// TIA Portal V18 export
FUNCTION_BLOCK "Control_Buttons_Activation"   // FB23, LAD
{ S7_Optimized_Access := 'TRUE' }
VERSION : 0.1
// stored: AutoNumber true, IsIECCheckEnabled false, IsRetainMemResEnabled false, MemoryReserve 100, SetENOAutomatically false, UDAEnableTagReadback false
   VAR_INPUT
      JogInZ1pos : Bool;
      JogInZ1neg : Bool;
      JogInZ2pos : Bool;
      JogInZ2neg : Bool;
   END_VAR
   VAR_OUTPUT
      Control_Buttons_Move_Permission : Bool;
      Control_Buttons_ActivatedOUT : Bool;
   END_VAR
   VAR
      Step01 : Bool;
      Step02 : Bool;
      Step03 : Bool;
      Step04 : Bool;
      Step05 : Bool;
      Step06 : Bool;
      Step07 : Bool;
      Step08 : Bool;
      AnyButtonPressed : Bool;
      AllButtonsPressed : Bool;
      ControlButtonsActivated : Bool;
   END_VAR
BEGIN

REGION Network 1: Any Button Pressed
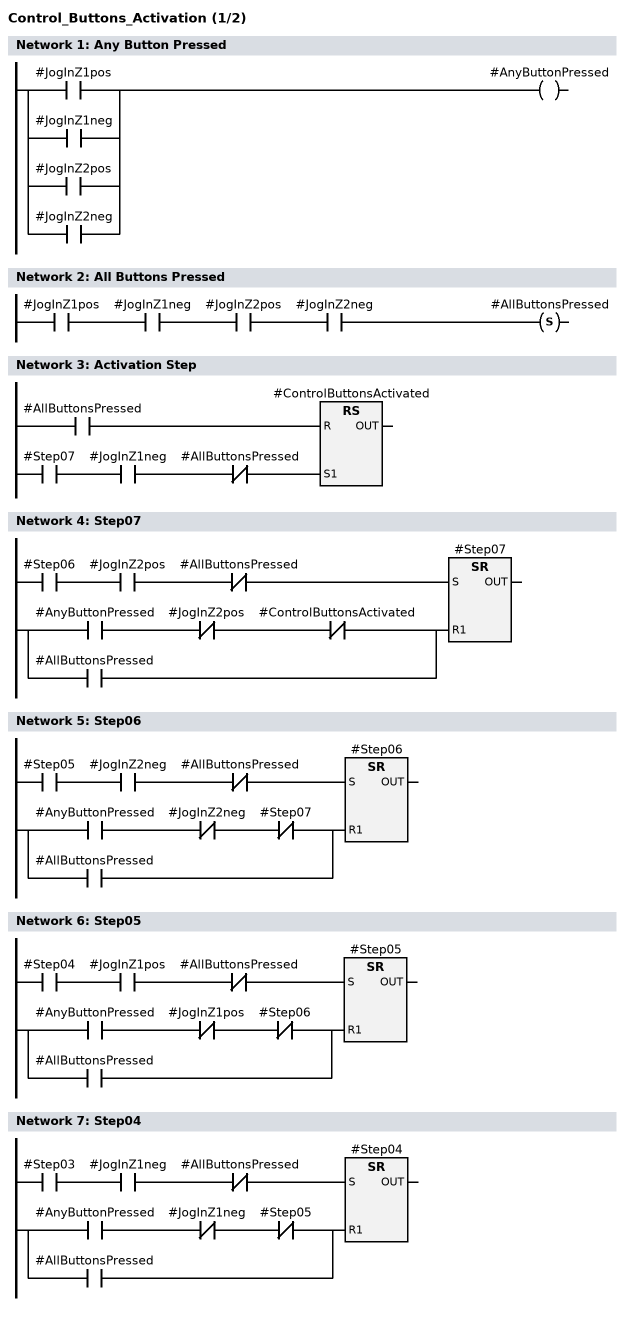
   RUNG wire#powerrail
      Contact( #JogInZ1pos )
      wire#w1
      Coil( #AnyButtonPressed )
   END_RUNG
   RUNG wire#powerrail
      Contact( #JogInZ1neg )
   END_RUNG wire#w1
   RUNG wire#powerrail
      Contact( #JogInZ2pos )
   END_RUNG wire#w1
   RUNG wire#powerrail
      Contact( #JogInZ2neg )
   END_RUNG wire#w1
   // the same network as SCL:
   #AnyButtonPressed := #JogInZ1pos OR #JogInZ1neg OR #JogInZ2pos OR #JogInZ2neg;
END_REGION

REGION Network 2: All Buttons Pressed
   RUNG wire#powerrail
      Contact( #JogInZ1pos )
      Contact( #JogInZ1neg )
      Contact( #JogInZ2pos )
      Contact( #JogInZ2neg )
      S_Coil( #AllButtonsPressed )
   END_RUNG
   // the same network as SCL:
   IF #JogInZ1pos AND #JogInZ1neg AND #JogInZ2pos AND #JogInZ2neg THEN #AllButtonsPressed := TRUE; END_IF;
END_REGION

REGION Network 3: Activation Step
   RUNG wire#powerrail
      Contact( #AllButtonsPressed )
      S_RS(operand := #ControlButtonsActivated, s1 := wire#w1)
   END_RUNG
   RUNG wire#powerrail
      Contact( #Step07 )
      Contact( #JogInZ1neg )
      I_Contact( #AllButtonsPressed )
   END_RUNG wire#w1
   // the same network as SCL:
   IF #AllButtonsPressed THEN
       #ControlButtonsActivated := FALSE;   // RS flip-flop
   END_IF;
   IF #Step07 AND #JogInZ1neg AND NOT #AllButtonsPressed THEN #ControlButtonsActivated := TRUE; END_IF;
END_REGION

REGION Network 4: Step07
   RUNG wire#powerrail
      Contact( #Step06 )
      Contact( #JogInZ2pos )
      I_Contact( #AllButtonsPressed )
      S_SR(operand := #Step07, r1 := wire#w1)
   END_RUNG
   RUNG wire#powerrail
      Contact( #AnyButtonPressed )
      I_Contact( #JogInZ2pos )
      I_Contact( #ControlButtonsActivated )
   END_RUNG wire#w1
   RUNG wire#powerrail
      Contact( #AllButtonsPressed )
   END_RUNG wire#w1
   // the same network as SCL:
   IF #Step06 AND #JogInZ2pos AND NOT #AllButtonsPressed THEN
       #Step07 := TRUE;   // SR flip-flop
   END_IF;
   IF (#AnyButtonPressed AND NOT #JogInZ2pos AND NOT #ControlButtonsActivated) OR #AllButtonsPressed THEN
       #Step07 := FALSE;
   END_IF;
END_REGION

REGION Network 5: Step06
   RUNG wire#powerrail
      Contact( #Step05 )
      Contact( #JogInZ2neg )
      I_Contact( #AllButtonsPressed )
      S_SR(operand := #Step06, r1 := wire#w1)
   END_RUNG
   RUNG wire#powerrail
      Contact( #AnyButtonPressed )
      I_Contact( #JogInZ2neg )
      I_Contact( #Step07 )
   END_RUNG wire#w1
   RUNG wire#powerrail
      Contact( #AllButtonsPressed )
   END_RUNG wire#w1
   // the same network as SCL:
   IF #Step05 AND #JogInZ2neg AND NOT #AllButtonsPressed THEN
       #Step06 := TRUE;   // SR flip-flop
   END_IF;
   IF (#AnyButtonPressed AND NOT #JogInZ2neg AND NOT #Step07) OR #AllButtonsPressed THEN
       #Step06 := FALSE;
   END_IF;
END_REGION

REGION Network 6: Step05
   RUNG wire#powerrail
      Contact( #Step04 )
      Contact( #JogInZ1pos )
      I_Contact( #AllButtonsPressed )
      S_SR(operand := #Step05, r1 := wire#w1)
   END_RUNG
   RUNG wire#powerrail
      Contact( #AnyButtonPressed )
      I_Contact( #JogInZ1pos )
      I_Contact( #Step06 )
   END_RUNG wire#w1
   RUNG wire#powerrail
      Contact( #AllButtonsPressed )
   END_RUNG wire#w1
   // the same network as SCL:
   IF #Step04 AND #JogInZ1pos AND NOT #AllButtonsPressed THEN
       #Step05 := TRUE;   // SR flip-flop
   END_IF;
   IF (#AnyButtonPressed AND NOT #JogInZ1pos AND NOT #Step06) OR #AllButtonsPressed THEN
       #Step05 := FALSE;
   END_IF;
END_REGION

REGION Network 7: Step04
   RUNG wire#powerrail
      Contact( #Step03 )
      Contact( #JogInZ1neg )
      I_Contact( #AllButtonsPressed )
      S_SR(operand := #Step04, r1 := wire#w1)
   END_RUNG
   RUNG wire#powerrail
      Contact( #AnyButtonPressed )
      I_Contact( #JogInZ1neg )
      I_Contact( #Step05 )
   END_RUNG wire#w1
   RUNG wire#powerrail
      Contact( #AllButtonsPressed )
   END_RUNG wire#w1
   // the same network as SCL:
   IF #Step03 AND #JogInZ1neg AND NOT #AllButtonsPressed THEN
       #Step04 := TRUE;   // SR flip-flop
   END_IF;
   IF (#AnyButtonPressed AND NOT #JogInZ1neg AND NOT #Step05) OR #AllButtonsPressed THEN
       #Step04 := FALSE;
   END_IF;
END_REGION

REGION Network 8: Step03
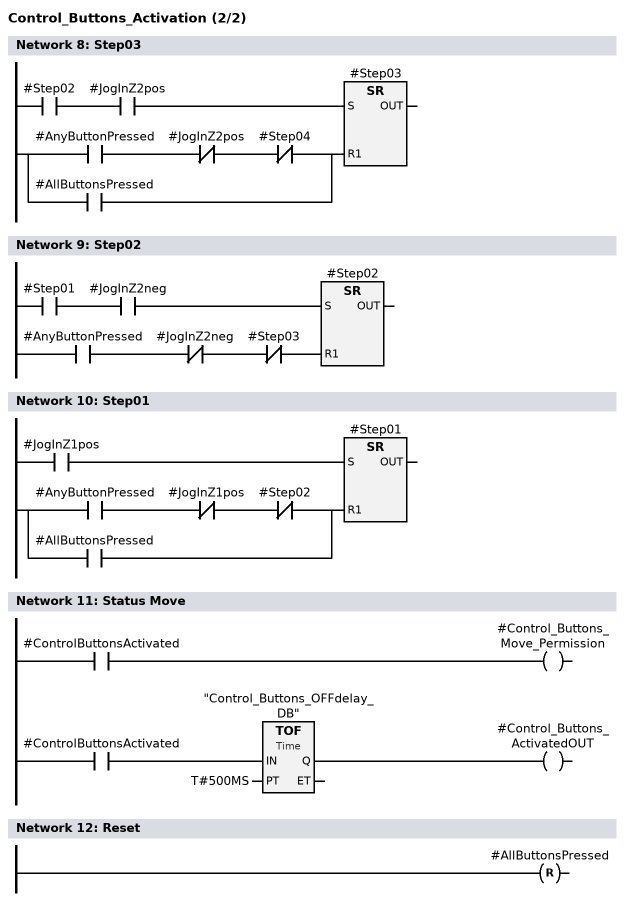
   RUNG wire#powerrail
      Contact( #Step02 )
      Contact( #JogInZ2pos )
      S_SR(operand := #Step03, r1 := wire#w1)
   END_RUNG
   RUNG wire#powerrail
      Contact( #AnyButtonPressed )
      I_Contact( #JogInZ2pos )
      I_Contact( #Step04 )
   END_RUNG wire#w1
   RUNG wire#powerrail
      Contact( #AllButtonsPressed )
   END_RUNG wire#w1
   // the same network as SCL:
   IF #Step02 AND #JogInZ2pos THEN
       #Step03 := TRUE;   // SR flip-flop
   END_IF;
   IF (#AnyButtonPressed AND NOT #JogInZ2pos AND NOT #Step04) OR #AllButtonsPressed THEN
       #Step03 := FALSE;
   END_IF;
END_REGION

REGION Network 9: Step02
   RUNG wire#powerrail
      Contact( #Step01 )
      Contact( #JogInZ2neg )
      S_SR(operand := #Step02, r1 := wire#w1)
   END_RUNG
   RUNG wire#powerrail
      Contact( #AnyButtonPressed )
      I_Contact( #JogInZ2neg )
      I_Contact( #Step03 )
   END_RUNG wire#w1
   // the same network as SCL:
   IF #Step01 AND #JogInZ2neg THEN
       #Step02 := TRUE;   // SR flip-flop
   END_IF;
   IF #AnyButtonPressed AND NOT #JogInZ2neg AND NOT #Step03 THEN #Step02 := FALSE; END_IF;
END_REGION

REGION Network 10: Step01
   RUNG wire#powerrail
      Contact( #JogInZ1pos )
      S_SR(operand := #Step01, r1 := wire#w1)
   END_RUNG
   RUNG wire#powerrail
      Contact( #AnyButtonPressed )
      I_Contact( #JogInZ1pos )
      I_Contact( #Step02 )
   END_RUNG wire#w1
   RUNG wire#powerrail
      Contact( #AllButtonsPressed )
   END_RUNG wire#w1
   // the same network as SCL:
   IF #JogInZ1pos THEN
       #Step01 := TRUE;   // SR flip-flop
   END_IF;
   IF (#AnyButtonPressed AND NOT #JogInZ1pos AND NOT #Step02) OR #AllButtonsPressed THEN
       #Step01 := FALSE;
   END_IF;
END_REGION

REGION Network 11: Status Move
   RUNG wire#powerrail
      Contact( #ControlButtonsActivated )
      Coil( #Control_Buttons_Move_Permission )
   END_RUNG
   RUNG wire#powerrail
      Contact( #ControlButtonsActivated )
      { S7_Templates := "time_type := Time" } "Control_Buttons_OFFdelay_DB".TOF(pt := T#500MS, et =>)
      Coil( #Control_Buttons_ActivatedOUT )
   END_RUNG
   // the same network as SCL:
   #Control_Buttons_Move_Permission := #ControlButtonsActivated;
   "Control_Buttons_OFFdelay_DB".TOF(IN := #ControlButtonsActivated, PT := T#500MS);
   #Control_Buttons_ActivatedOUT := "Control_Buttons_OFFdelay_DB".Q;
END_REGION

REGION Network 12: Reset
   RUNG wire#powerrail
      R_Coil( #AllButtonsPressed )
   END_RUNG
   // the same network as SCL:
   #AllButtonsPressed := FALSE;
END_REGION
END_FUNCTION_BLOCK
